(* Schneider Machine Expert - Basic project water_pump_realpars_LD, file version 2.7.0.0 *)
(* ProjectInformations: Name=New project *)

HARDWARE
  Cpu 0: TM221M16R/G
  EthernetConfiguration: NetworkName=M221, IpAllocationMode=FixedAddress, IpAddress=0.0.0.0, SubnetMask=0.0.0.0
  SerialLineConfiguration: Baud=Baud19200, Parity=ParityEven, DataBits=DataBits8, StopBits=StopBits1, PhysicalMedium=PhysicalMediumRs485, TransmissionMode=TransmissionModeModbusRtu, SlaveId=1, Addressing=SlaveAddressing
  MastTask: UsePeriodScanMode=false, PeriodScan=100
  FastTask: Period=255
  CpuBehavior: StartingMode=StartAsPreviousState, AutoSaveRamOnEeprom=true, WatchdogPeriod=250

SYMBOLS  (address, symbol, comment, settings)
  %TM1        [Type=TP, Preset=7, Base=OneSecond]
  %I0.0     STARTED
  %I0.1     STOP
  %I0.2     LLS
  %I0.3     HLS
  %Q0.0     PUMP1
  %Q0.1     PUMP2
  %Q0.2     MIXER
  %Q0.3     VALVE

POU pump1
  (* SectionNumber=1 *)

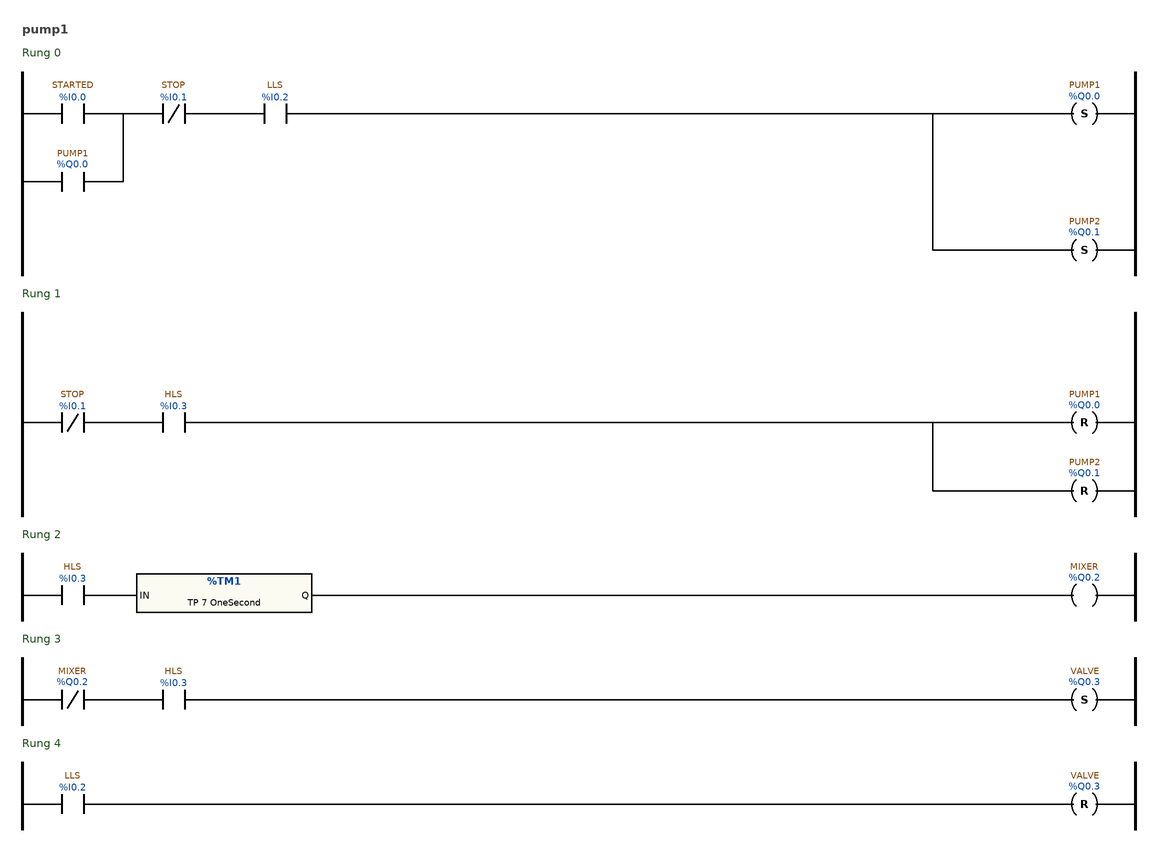

// Rung 0
  LD %I0.0                (* STARTED *)
  OR %Q0.0                (* PUMP1 *)
  ANDN %I0.1              (* STOP *)
  AND %I0.2               (* LLS *)
  S %Q0.0                 (* PUMP1 *)
  S %Q0.1                 (* PUMP2 *)
  // as ST:
  //   _t1 := (STARTED OR PUMP1) AND NOT STOP AND LLS;
  //   IF _t1 THEN PUMP1 := TRUE; END_IF;
  //   IF _t1 THEN PUMP2 := TRUE; END_IF;

// Rung 1
  LDN %I0.1               (* STOP *)
  AND %I0.3               (* HLS *)
  R %Q0.0                 (* PUMP1 *)
  R %Q0.1                 (* PUMP2 *)
  // as ST:
  //   IF NOT STOP AND HLS THEN PUMP1 := FALSE; END_IF;
  //   IF NOT STOP AND HLS THEN PUMP2 := FALSE; END_IF;

// Rung 2
  BLK %TM1
  LD %I0.3                (* HLS *)
  IN
  OUT_BLK
  LD Q
  ST %Q0.2                (* MIXER *)
  END_BLK
  // as ST:
  //   %TM1(IN := HLS);
  //   MIXER := %TM1.Q;

// Rung 3
  LDN %Q0.2               (* MIXER *)
  AND %I0.3               (* HLS *)
  S %Q0.3                 (* VALVE *)
  // as ST:
  //   IF NOT MIXER AND HLS THEN VALVE := TRUE; END_IF;

// Rung 4
  LD %I0.2                (* LLS *)
  R %Q0.3                 (* VALVE *)
  // as ST:
  //   IF LLS THEN VALVE := FALSE; END_IF;
